Staubli VAL3: Exam_2025_59333.dtx

mdesc mNomSpeed
mdesc mRapide = {accel=75, vel=75, decel=75}
mdesc mLent = {accel=10, vel=10, decel=10}
pointRx pP1 = {fatherId=world[0]}
jointRx jDepart
num nDistancePiece = 80
num nDistanceLigne = 160
num nPieceLigne = 3
num nLigne
bool bDCY = true
num nHauteurPiece = 100
tool tPince = {z=100, fatherId=flange[0], ioLink=valve1}
trsf trAppro = {z=-100}
trsf trDecalPiece
trsf trDecalHauteur
num nCycles
num nDebut
num nFin
